// TIA Portal V17 export
// export: Created 2022-07-20T07:02:39.0698201Z, ExportSetting WithDefaults, DisplayName Totally Integrated Automation Portal, DisplayVersion V17, DisplayName TIA Portal Openness, DisplayVersion V17, DisplayName TIA Portal Version Control Interface, DisplayVersion V17, DisplayName SINAMICS Startdrive Advanced, DisplayVersion V17, DisplayName SINAMICS Startdrive G130, G150, S120, S150, SINAMICS MV, S210, DisplayVersion V17, DisplayName SINAMICS Startdrive G110M, G120, G120C, G120D, G120P, G115D, DisplayVersion V17, DisplayName STEP 7 Professional, DisplayVersion V17, DisplayName STEP 7 Safety, DisplayVersion V17, DisplayName WinCC Advanced, DisplayVersion V17
VAR_GLOBAL   // PLC tag table "Pilz_CommmunicationTable"
   Pilz_OutputByte0_1 AT %QB1000 : Byte;
   Pilz_OutputByte0_2 AT %QB1001 : Byte;
   Pilz_OutputByte0_3 AT %QB1002 : Byte;
   Pilz_OutputByte0_4 AT %QB1003 : Byte;
   Pilz_OutputByte1_1 AT %QB1004 : Byte;
   Pilz_OutputByte1_2 AT %QB1005 : Byte;
   Pilz_OutputByte1_3 AT %QB1006 : Byte;
   Pilz_OutputByte1_4 AT %QB1007 : Byte;
   Pilz_OutputByte2_1 AT %QB1008 : Byte;
   Pilz_OutputByte2_2 AT %QB1009 : Byte;
   Pilz_OutputByte2_3 AT %QB1010 : Byte;
   Pilz_OutputByte2_4 AT %QB1011 : Byte;
   Pilz_OutputByte3_1 AT %QB1012 : Byte;
   Pilz_OutputByte3_2 AT %QB1013 : Byte;
   Pilz_OutputByte3_3 AT %QB1014 : Byte;
   Pilz_OutputByte3_4 AT %QB1015 : Byte;
   Pilz_InputByte0_1 AT %IB1000 : Byte;
   Pilz_InputByte0_2 AT %IB1001 : Byte;
   Pilz_InputByte0_3 AT %IB1002 : Byte;
   Pilz_InputByte0_4 AT %IB1003 : Byte;
   Pilz_InputByte1_1 AT %IB1004 : Byte;
   Pilz_InputByte1_2 AT %IB1005 : Byte;
   Pilz_InputByte1_3 AT %IB1006 : Byte;
   Pilz_InputByte1_4 AT %IB1007 : Byte;
   Pilz_InputByte2_1 AT %IB1008 : Byte;
   Pilz_InputByte2_2 AT %IB1009 : Byte;
   Pilz_InputByte2_3 AT %IB1010 : Byte;
   Pilz_InputByte2_4 AT %IB1011 : Byte;
   Pilz_InputByte3_1 AT %IB1012 : Byte;
   Pilz_InputByte3_2 AT %IB1013 : Byte;
   Pilz_InputByte3_3 AT %IB1014 : Byte;
   Pilz_InputByte3_4 AT %IB1015 : Byte;
END_VAR
